RoboDK station: KR10 08222019 Plank print plz dont break.rdk

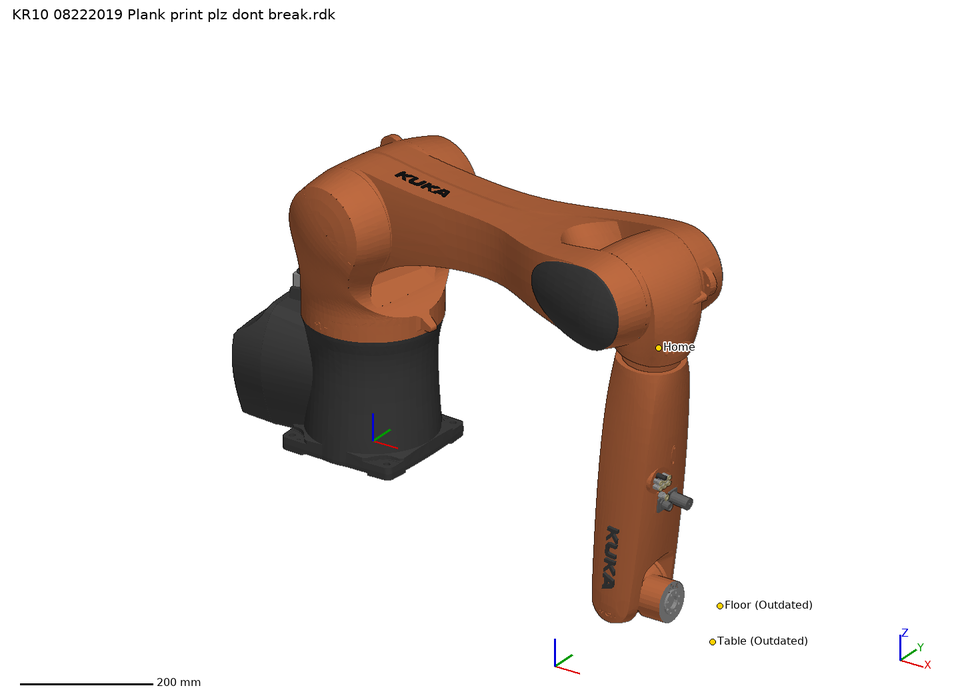
[picture v0: the station drawn from its stored meshes, robots at their saved joint values, targets as dots, program paths as lines]
Station KR10 08222019 Plank print plz dont break. Poses are relative to the parent item; angles as X-Y-Z fixed-axis rotations.
  - frame KUKA KR 10 R1100 sixx Base at (0, 0, 0) mm
    - robot KUKA KR 10 R1100 sixx: 6 axes, payload 10 kg, reach 1101 mm, repeatability 0.03 mm, weight 54 kg
        modified DH rows (alpha deg, a mm, theta deg, d mm): 0, 0, 0, 400; -90, 25, 0, 0; 0, 560, -90, 0; -90, 35, 0, 515; 90, 0, 0, 0; -90, 0, 180, 80
        joint limits [-170, -190, -120, -185, -120, -350] to [170, 45, 156, 185, 120, 350]; home [0, -90, 90, 0, 0, 0]; saved at [11.031, -6.458, 102.945, 11.1, -96.367, -18.611]
      - tool Tool 1, TCP at (63, 0, 57) mm, rotated rx 0 ry 0 rz -19.86 deg
    - target Home (joint target) at (585.45, -85.67, 353.51) mm, rotated rx 0 ry 90 rz 0 deg; joints [10.816, -63.304, 136.787, 11.27, -73.784, -3.185] of KUKA KR 10 R1100 sixx
    - target Floor (Outdated) (Cartesian target) at (689.85, -72.33, -55.42) mm, rotated rx 0 ry 78 rz 0 deg; joints [8.166, -9.123, 106.388, 8.491, -110.738, -3.85] of KUKA KR 10 R1100 sixx
    - target Table (Outdated) (Cartesian target) at (684.73, -85.37, -111.93) mm, rotated rx -154.84 ry 90 rz -154.84 deg; joints [9.441, -6.412, 103.401, 9.542, -98.443, -3.794] of KUKA KR 10 R1100 sixx
  - frame Plank bed at (570.65, -336.33, -83.6) mm, rotated rx 0.03 ry -0.06 rz 0 deg
